TYPE Vessel :
STRUCT
	LLS : BOOL;	
	ULS : BOOL;	
	
	Valves : ARRAY[0..7] OF Valve;
	Pumps : ARRAY[0..1] OF Pump; 
//	VentValve : Valve;
//	N2PurgeValve : Valve;
//	TransferValve : Valve;
//	FillInValve : Valve;
//	FillInHeaderValve : Valve;
// 	DrainValve : Valve;
//	FlushingValve : Valve;

//	FillInPump : PUMP;
//	TransferPump : PUMP;
	
	
	
END_STRUCT
END_TYPE

(* stored: Version 1.1.0.1, ProductVersion 3.1.4024.3
   DUT Vessel: Id {bd272d08-88e2-4cd5-872e-6421638a2e1c} *)
